// TIA Portal V15.1 export
// export: Created 2024-06-21T08:41:06.7682884Z, ExportSetting WithDefaults, DisplayName Totally Integrated Automation Portal, DisplayVersion V15.1 Update 5, DisplayName TIA Portal Openness, DisplayVersion V15.1 Update 5, DisplayName SINAMICS Startdrive Advanced, DisplayVersion V15.1, DisplayName G130, G150, S120, S150, SINAMICS MV, S210, DisplayVersion V15.1, DisplayName G110M, G120, G120C, G120D, G120P, DisplayVersion V15.1, DisplayName STEP 7 Professional, DisplayVersion V15.1 Update 5, DisplayName STEP 7 Safety, DisplayVersion V15.1, DisplayName WinCC Professional, DisplayVersion V15.1 Update 5, DisplayName SIMATIC Visualization Architect, DisplayVersion V15.1
FUNCTION_BLOCK "LGBBeltControl"   // FB6632, FBD
TITLE = LAcofDet / LGBBeltControl
{ S7_Optimized_Access := 'TRUE' }
AUTHOR : VCC
FAMILY : AlarmHandling
NAME : LGBBeltControl
VERSION : 1.0
// ===============================================================================
// This module handles a partdetection with all his functions and alarms
// Functions are DetCheckOn, DetCheckOff and EnableAlarm
// Outputs are DetAlarm and DetSim signal
// ===============================================================================
// ============================================================================
// This module handles Belt Slip Control
// ============================================================================
// stored: AutoNumber false, IsIECCheckEnabled false, IsRetainMemResEnabled false, MemoryReserve 100, SetENOAutomatically False, UDAEnableTagReadback false
   VAR_INPUT
      I_Det1SlipCtrl { ExternalAccessible := 'False'; ExternalVisible := 'False'; ExternalWritable := 'False'} : Bool;   // Actual input from sensor
      I_Det2SlipCtrl { ExternalAccessible := 'False'; ExternalVisible := 'False'; ExternalWritable := 'False'} : Bool;   // Actual input from sensor
      I_MotorRunning { ExternalAccessible := 'False'; ExternalVisible := 'False'; ExternalWritable := 'False'} : Bool;   // Previous detection
      I_EnableAlarm { ExternalAccessible := 'False'; ExternalVisible := 'False'; ExternalWritable := 'False'} : Bool;   // Enable Alarm
      I_AlarmClass { ExternalAccessible := 'False'; ExternalVisible := 'False'; ExternalWritable := 'False'} : Char;   // Alarm class -> A - B - C - D or E
      I_AlarmResetPB { ExternalAccessible := 'False'; ExternalVisible := 'False'; ExternalWritable := 'False'} : Bool;   // Alarm reset pushbutton is activated
   END_VAR
   VAR_OUTPUT
      O_Alarm { ExternalAccessible := 'False'; ExternalVisible := 'False'; ExternalWritable := 'False'} : Bool;   // Detection ON too long alarm / Detection alarm
      O_AlarmABCondition { ExternalAccessible := 'False'; ExternalVisible := 'False'; ExternalWritable := 'False'} : Bool;   // Alarm AB condition
   END_VAR
   VAR_IN_OUT
      H_HMI : "H_HMI";   // H_HMI
      H_BeltControl : "H_GBBeltControl";   // H_KTLBeltSlipControl
      IO_Modes : "Modes";
   END_VAR
   VAR
      CounterSlipCtrl { ExternalAccessible := 'False'; ExternalVisible := 'False'; ExternalWritable := 'False'} : DInt;   // Counter Slip Control
      CounterSlipCtrlL { ExternalAccessible := 'False'; ExternalVisible := 'False'; ExternalWritable := 'False'} : DInt;   // Counter Slip Control Left
      CounterSlipCtrlR { ExternalAccessible := 'False'; ExternalVisible := 'False'; ExternalWritable := 'False'} : DInt;   // Counter Slip Control Right
      AbsCounterSlipCtrl { ExternalAccessible := 'False'; ExternalVisible := 'False'; ExternalWritable := 'False'} : DInt;   // ABS Counter Slip Control
      ResetCount { ExternalAccessible := 'False'; ExternalVisible := 'False'; ExternalWritable := 'False'} : Bool;   // Reset Counters
      AlarmCond { ExternalAccessible := 'False'; ExternalVisible := 'False'; ExternalWritable := 'False'} : Bool;   // Alarm condition / Static variable of O_DetAlarm
      AlarmCondNOCountL { ExternalAccessible := 'False'; ExternalVisible := 'False'; ExternalWritable := 'False'} : Bool;   // Alarm condition / Static variable of O_DetAlarm
      AlarmCondNOCountR { ExternalAccessible := 'False'; ExternalVisible := 'False'; ExternalWritable := 'False'} : Bool;   // Alarm condition / Static variable of O_DetAlarm
      AlarmCondNCCountL { ExternalAccessible := 'False'; ExternalVisible := 'False'; ExternalWritable := 'False'} : Bool;   // Alarm condition / Static variable of O_DetAlarm
      AlarmCondNCCountR { ExternalAccessible := 'False'; ExternalVisible := 'False'; ExternalWritable := 'False'} : Bool;   // Alarm condition / Static variable of O_DetAlarm
      Alarm { ExternalAccessible := 'False'; ExternalVisible := 'False'; ExternalWritable := 'False'} : Bool;   // Alarm / Alarm condition
      AlarmClass_A { ExternalAccessible := 'False'; ExternalVisible := 'False'; ExternalWritable := 'False'} : Bool;   // The alarm is from alarm class A
      AlarmClass_B { ExternalAccessible := 'False'; ExternalVisible := 'False'; ExternalWritable := 'False'} : Bool;   // The alarm is from alarm class B
      AlarmClass_C { ExternalAccessible := 'False'; ExternalVisible := 'False'; ExternalWritable := 'False'} : Bool;   // The alarm is from alarm class C
      AlarmClass_D { ExternalAccessible := 'False'; ExternalVisible := 'False'; ExternalWritable := 'False'} : Bool;   // The alarm is from alarm class D
      AlarmClass_E { ExternalAccessible := 'False'; ExternalVisible := 'False'; ExternalWritable := 'False'} : Bool := false;   // The alarm is from alarm class E
      AlarmFiltered { ExternalAccessible := 'False'; ExternalVisible := 'False'; ExternalWritable := 'False'} : Bool;
      _TimerNoCountL { ExternalAccessible := 'False'; ExternalVisible := 'False'; ExternalWritable := 'False'} : "LTimer";
      _TimerNoCountR { ExternalAccessible := 'False'; ExternalVisible := 'False'; ExternalWritable := 'False'} : "LTimer";
      _TimerNcCountL { ExternalAccessible := 'False'; ExternalVisible := 'False'; ExternalWritable := 'False'} : "LTimer";
      _TimerNcCountR { ExternalAccessible := 'False'; ExternalVisible := 'False'; ExternalWritable := 'False'} : "LTimer";
      _TimerResetCount { ExternalAccessible := 'False'; ExternalVisible := 'False'; ExternalWritable := 'False'} : "LTimer";
      _TimerAlarmFilter { ExternalAccessible := 'False'; ExternalVisible := 'False'; ExternalWritable := 'False'} : "LTimer";
      edge { ExternalAccessible := 'False'; ExternalVisible := 'False'; ExternalWritable := 'False'} : Array[0..1] of Bool;
   END_VAR
   VAR_TEMP   // added for the SCL form of the ladder/FBD networks
      _w1 : Bool;
      _w2 : Bool;
   END_VAR
BEGIN

REGION Network 1: **** 1 - Inputs **** HMI Commands
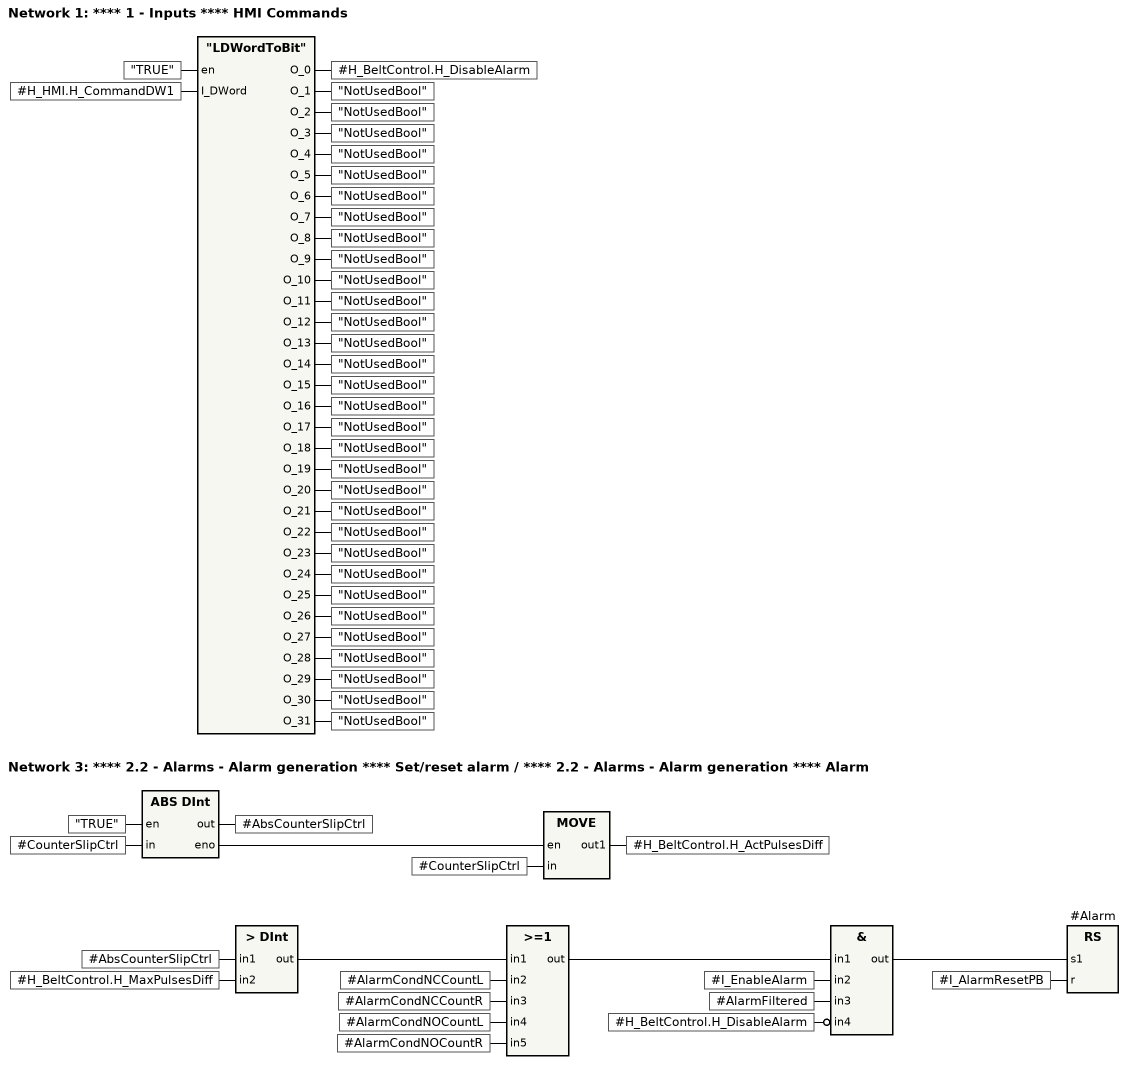
   IF "TRUE" THEN
       "LDWordToBit"(I_DWord := #H_HMI.H_CommandDW1,
                     O_0 => #H_BeltControl.H_DisableAlarm,
                     O_1 => "NotUsedBool",
                     O_2 => "NotUsedBool",
                     O_3 => "NotUsedBool",
                     O_4 => "NotUsedBool",
                     O_5 => "NotUsedBool",
                     O_6 => "NotUsedBool",
                     O_7 => "NotUsedBool",
                     O_8 => "NotUsedBool",
                     O_9 => "NotUsedBool",
                     O_10 => "NotUsedBool",
                     O_11 => "NotUsedBool",
                     O_12 => "NotUsedBool",
                     O_13 => "NotUsedBool",
                     O_14 => "NotUsedBool",
                     O_15 => "NotUsedBool",
                     O_16 => "NotUsedBool",
                     O_17 => "NotUsedBool",
                     O_18 => "NotUsedBool",
                     O_19 => "NotUsedBool",
                     O_20 => "NotUsedBool",
                     O_21 => "NotUsedBool",
                     O_22 => "NotUsedBool",
                     O_23 => "NotUsedBool",
                     O_24 => "NotUsedBool",
                     O_25 => "NotUsedBool",
                     O_26 => "NotUsedBool",
                     O_27 => "NotUsedBool",
                     O_28 => "NotUsedBool",
                     O_29 => "NotUsedBool",
                     O_30 => "NotUsedBool",
                     O_31 => "NotUsedBool");
   END_IF;
END_REGION

NETWORK
TITLE = **** 1 - Inputs **** Alarm class
// Alarm class
// Alarm class = E
      L     #I_AlarmClass;
      L     'E';
      ==I;
      =     #AlarmClass_E;

// Alarm class = D
      L     #I_AlarmClass;
      L     'D';
      ==I;
      =     #AlarmClass_D;

// Alarm class = C
      L     #I_AlarmClass;
      L     'C';
      ==I;
      =     #AlarmClass_C;

// Alarm class = B
      L     #I_AlarmClass;
      L     'B';
      ==I;
      =     #AlarmClass_B;

// Alarm class = A
      AN    #AlarmClass_B;
      AN    #AlarmClass_C;
      AN    #AlarmClass_D;
      AN    #AlarmClass_E;
      =     #AlarmClass_A;


REGION Network 3: **** 2.2 - Alarms - Alarm generation **** Set/reset alarm / **** 2.2 - Alarms - Alarm generation **** Alarm
   // Set/reset alarm
   IF "TRUE" THEN
       #AbsCounterSlipCtrl := ABS(#CounterSlipCtrl);
       #H_BeltControl.H_ActPulsesDiff := #CounterSlipCtrl;
   END_IF;
   IF #I_AlarmResetPB THEN
       #Alarm := FALSE;   // RS flip-flop
   END_IF;
   IF ((#AbsCounterSlipCtrl > #H_BeltControl.H_MaxPulsesDiff) OR #AlarmCondNCCountL OR #AlarmCondNCCountR OR #AlarmCondNOCountL OR #AlarmCondNOCountR) AND #I_EnableAlarm AND #AlarmFiltered AND NOT #H_BeltControl.H_DisableAlarm THEN
       #Alarm := TRUE;
   END_IF;
END_REGION

REGION Network 4: **** 2.2 - Alarms - Alarm generation **** Creating alarm overtime / **** 2.2 - Alarms - Alarm generation **** Pulses counters
   // Creating alarm overtime / Pulses counters
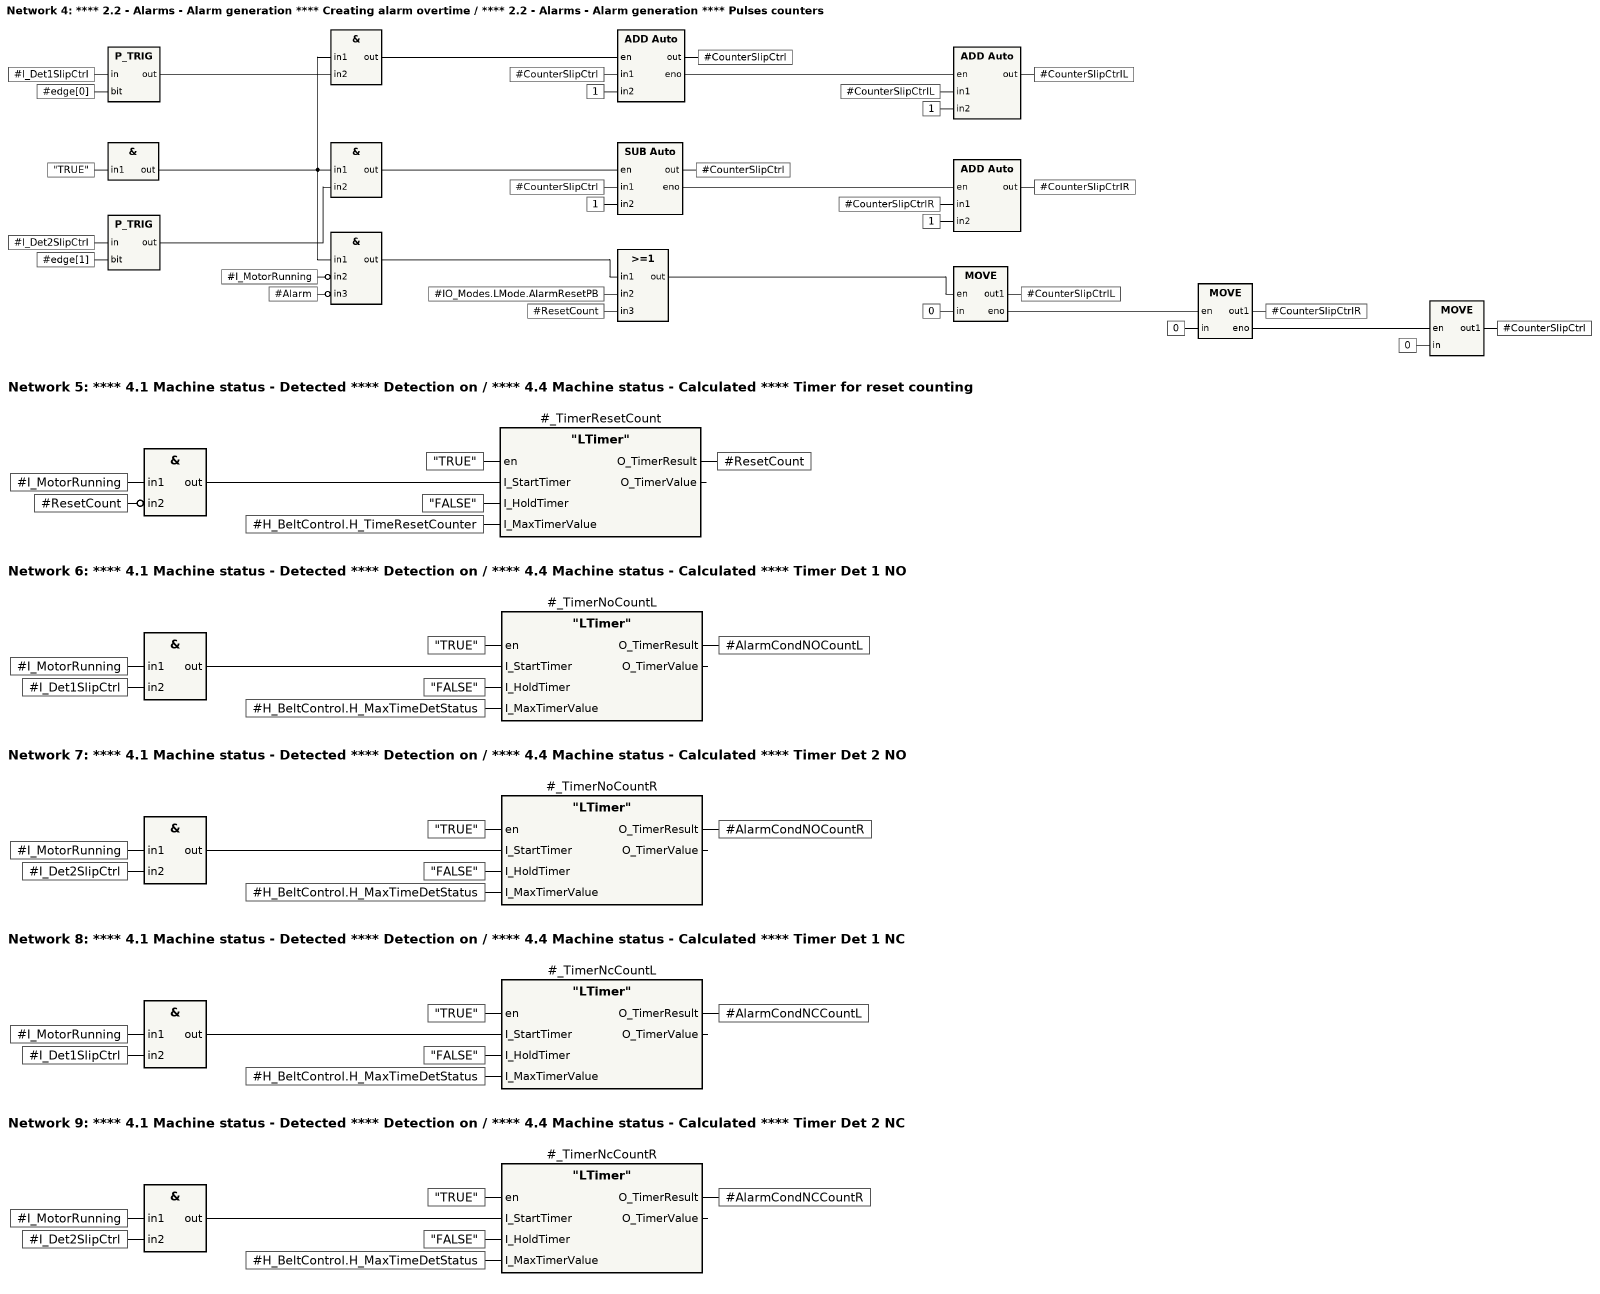
   #_w1 := #I_Det1SlipCtrl AND NOT #edge[0];   // rising edge
   #edge[0] := #I_Det1SlipCtrl;
   IF "TRUE" AND #_w1 THEN
       #CounterSlipCtrl := #CounterSlipCtrl + 1;
       #CounterSlipCtrlL := #CounterSlipCtrlL + 1;
   END_IF;
   #_w2 := #I_Det2SlipCtrl AND NOT #edge[1];   // rising edge
   #edge[1] := #I_Det2SlipCtrl;
   IF "TRUE" AND #_w2 THEN
       #CounterSlipCtrl := #CounterSlipCtrl - 1;
       #CounterSlipCtrlR := #CounterSlipCtrlR + 1;
   END_IF;
   IF ("TRUE" AND NOT #I_MotorRunning AND NOT #Alarm) OR #IO_Modes.LMode.AlarmResetPB OR #ResetCount THEN
       #CounterSlipCtrlL := 0;
       #CounterSlipCtrlR := 0;
       #CounterSlipCtrl := 0;
   END_IF;
END_REGION

REGION Network 5: **** 4.1 Machine status - Detected **** Detection on / **** 4.4 Machine status - Calculated **** Timer for reset counting
   // Detection on / Timer for reset counting
   IF "TRUE" THEN
       #_TimerResetCount(I_StartTimer := #I_MotorRunning AND NOT #ResetCount,   // "LTimer"
                         I_HoldTimer := "FALSE",
                         I_MaxTimerValue := #H_BeltControl.H_TimeResetCounter,
                         O_TimerResult => #ResetCount);
   END_IF;
END_REGION

REGION Network 6: **** 4.1 Machine status - Detected **** Detection on / **** 4.4 Machine status - Calculated **** Timer Det 1 NO
   // Detection on / Timer Det 1 NO
   IF "TRUE" THEN
       #_TimerNoCountL(I_StartTimer := #I_MotorRunning AND #I_Det1SlipCtrl,   // "LTimer"
                       I_HoldTimer := "FALSE",
                       I_MaxTimerValue := #H_BeltControl.H_MaxTimeDetStatus,
                       O_TimerResult => #AlarmCondNOCountL);
   END_IF;
END_REGION

REGION Network 7: **** 4.1 Machine status - Detected **** Detection on / **** 4.4 Machine status - Calculated **** Timer Det 2 NO
   // Detection on / Timer Det 2 NO
   IF "TRUE" THEN
       #_TimerNoCountR(I_StartTimer := #I_MotorRunning AND #I_Det2SlipCtrl,   // "LTimer"
                       I_HoldTimer := "FALSE",
                       I_MaxTimerValue := #H_BeltControl.H_MaxTimeDetStatus,
                       O_TimerResult => #AlarmCondNOCountR);
   END_IF;
END_REGION

REGION Network 8: **** 4.1 Machine status - Detected **** Detection on / **** 4.4 Machine status - Calculated **** Timer Det 1 NC
   // Detection on / Timer Det 1 NC
   IF "TRUE" THEN
       #_TimerNcCountL(I_StartTimer := #I_MotorRunning AND #I_Det1SlipCtrl,   // "LTimer"
                       I_HoldTimer := "FALSE",
                       I_MaxTimerValue := #H_BeltControl.H_MaxTimeDetStatus,
                       O_TimerResult => #AlarmCondNCCountL);
   END_IF;
END_REGION

REGION Network 9: **** 4.1 Machine status - Detected **** Detection on / **** 4.4 Machine status - Calculated **** Timer Det 2 NC
   // Detection on / Timer Det 2 NC
   IF "TRUE" THEN
       #_TimerNcCountR(I_StartTimer := #I_MotorRunning AND #I_Det2SlipCtrl,   // "LTimer"
                       I_HoldTimer := "FALSE",
                       I_MaxTimerValue := #H_BeltControl.H_MaxTimeDetStatus,
                       O_TimerResult => #AlarmCondNCCountR);
   END_IF;
END_REGION

REGION Network 10: **** 4.1 Machine status - Detected **** Detection on / **** 4.4 Machine status - Calculated **** Timer Alarm Filter
   // Detection on / Timer Det 2 NC
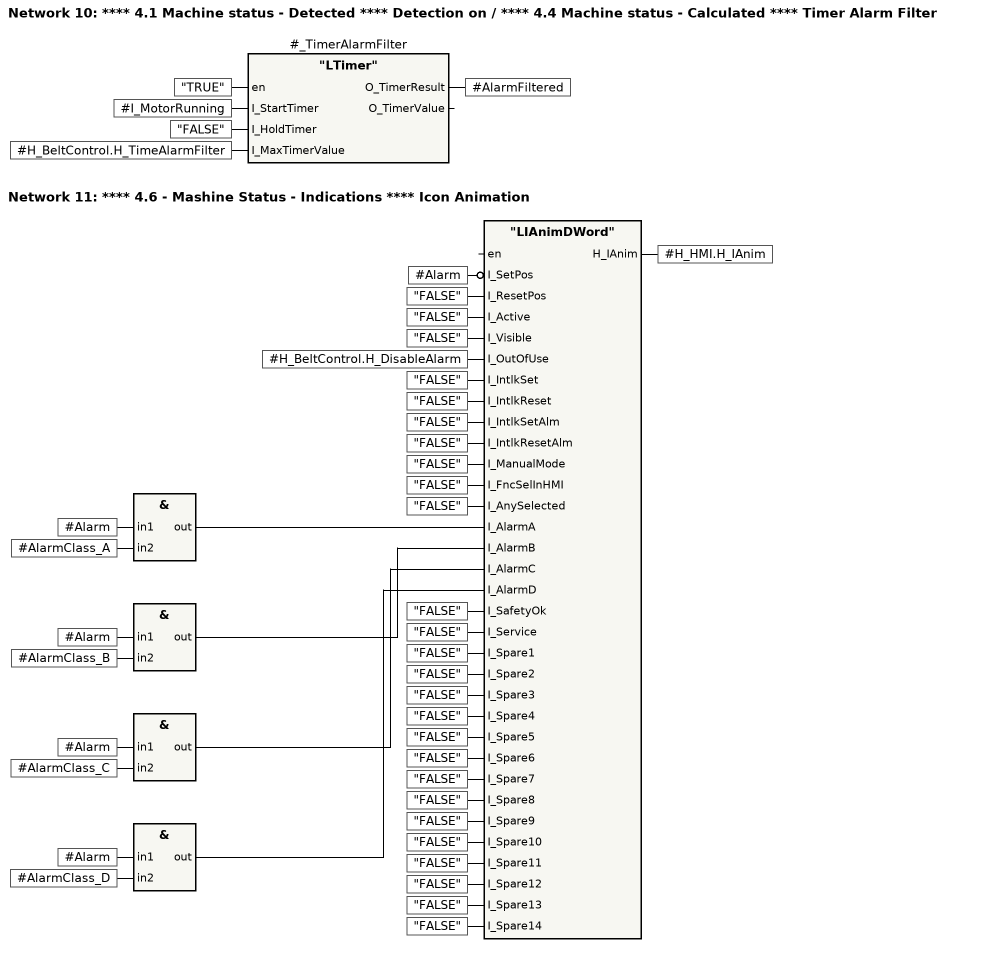
   IF "TRUE" THEN
       #_TimerAlarmFilter(I_StartTimer := #I_MotorRunning,   // "LTimer"
                          I_HoldTimer := "FALSE",
                          I_MaxTimerValue := #H_BeltControl.H_TimeAlarmFilter,
                          O_TimerResult => #AlarmFiltered);
   END_IF;
END_REGION

REGION Network 11: **** 4.6 - Mashine Status - Indications **** Icon Animation
   // Icon Animation
   "LIAnimDWord"(I_SetPos := NOT #Alarm,
                 I_ResetPos := "FALSE",
                 I_Active := "FALSE",
                 I_Visible := "FALSE",
                 I_OutOfUse := #H_BeltControl.H_DisableAlarm,
                 I_IntlkSet := "FALSE",
                 I_IntlkReset := "FALSE",
                 I_IntlkSetAlm := "FALSE",
                 I_IntlkResetAlm := "FALSE",
                 I_ManualMode := "FALSE",
                 I_FncSelInHMI := "FALSE",
                 I_AnySelected := "FALSE",
                 I_AlarmA := #Alarm AND #AlarmClass_A,
                 I_AlarmB := #Alarm AND #AlarmClass_B,
                 I_AlarmC := #Alarm AND #AlarmClass_C,
                 I_AlarmD := #Alarm AND #AlarmClass_D,
                 I_SafetyOk := "FALSE",
                 I_Service := "FALSE",
                 I_Spare1 := "FALSE",
                 I_Spare2 := "FALSE",
                 I_Spare3 := "FALSE",
                 I_Spare4 := "FALSE",
                 I_Spare5 := "FALSE",
                 I_Spare6 := "FALSE",
                 I_Spare7 := "FALSE",
                 I_Spare8 := "FALSE",
                 I_Spare9 := "FALSE",
                 I_Spare10 := "FALSE",
                 I_Spare11 := "FALSE",
                 I_Spare12 := "FALSE",
                 I_Spare13 := "FALSE",
                 I_Spare14 := "FALSE",
                 H_IAnim => #H_HMI.H_IAnim);
END_REGION

REGION Network 12: **** 4.6 - Machine Status - Indications **** Animation
   // Animation
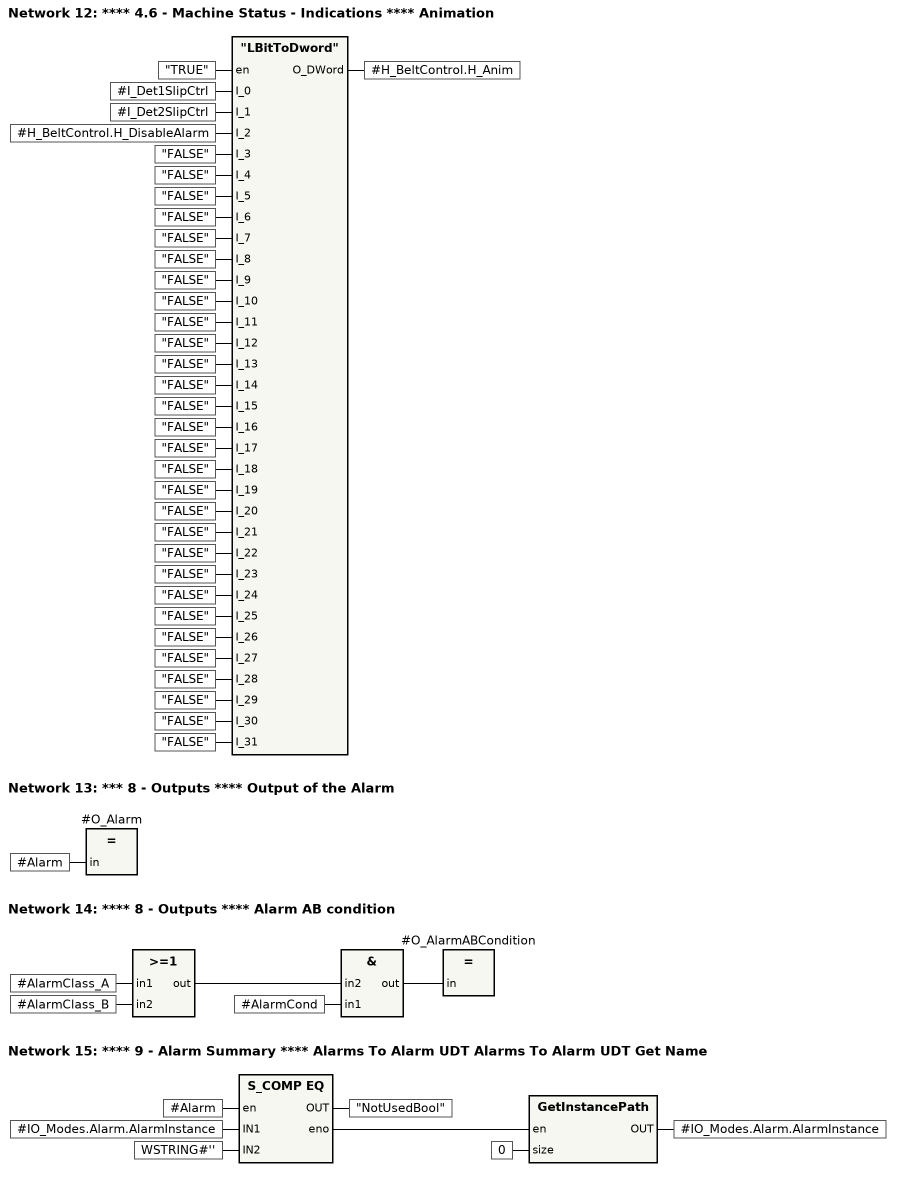
   IF "TRUE" THEN
       "LBitToDword"(I_0 := #I_Det1SlipCtrl,
                     I_1 := #I_Det2SlipCtrl,
                     I_2 := #H_BeltControl.H_DisableAlarm,
                     I_3 := "FALSE",
                     I_4 := "FALSE",
                     I_5 := "FALSE",
                     I_6 := "FALSE",
                     I_7 := "FALSE",
                     I_8 := "FALSE",
                     I_9 := "FALSE",
                     I_10 := "FALSE",
                     I_11 := "FALSE",
                     I_12 := "FALSE",
                     I_13 := "FALSE",
                     I_14 := "FALSE",
                     I_15 := "FALSE",
                     I_16 := "FALSE",
                     I_17 := "FALSE",
                     I_18 := "FALSE",
                     I_19 := "FALSE",
                     I_20 := "FALSE",
                     I_21 := "FALSE",
                     I_22 := "FALSE",
                     I_23 := "FALSE",
                     I_24 := "FALSE",
                     I_25 := "FALSE",
                     I_26 := "FALSE",
                     I_27 := "FALSE",
                     I_28 := "FALSE",
                     I_29 := "FALSE",
                     I_30 := "FALSE",
                     I_31 := "FALSE",
                     O_DWord => #H_BeltControl.H_Anim);
   END_IF;
END_REGION

REGION Network 13: *** 8 - Outputs **** Output of the Alarm
   // Output of the Alarm
   #O_Alarm := #Alarm;
END_REGION

REGION Network 14: **** 8 - Outputs **** Alarm AB condition
   // Alarm AB condition
   #O_AlarmABCondition := (#AlarmClass_A OR #AlarmClass_B) AND #AlarmCond;
END_REGION

REGION Network 15: **** 9 - Alarm Summary **** Alarms To Alarm UDT Alarms To Alarm UDT Get Name
   // Alarm / Alarm D
   S_COMP(EN := #Alarm,
          IN1 := #IO_Modes.Alarm.AlarmInstance,
          IN2 := WSTRING#'',
          OUT => "NotUsedBool",
          ENO => #_w1);
   IF #_w1 THEN GetInstancePath(size := 0, OUT => #IO_Modes.Alarm.AlarmInstance); END_IF;
END_REGION

REGION Network 16: **** 9 - Alarm Summary **** Alarms To Alarm UDT
   // Alarm / Alarm D
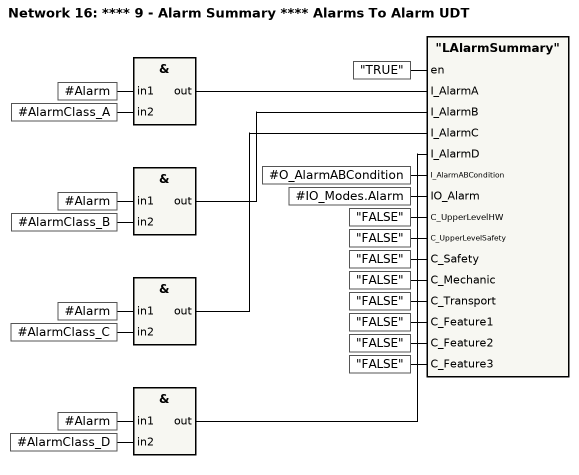
   IF "TRUE" THEN
       "LAlarmSummary"(I_AlarmA := #Alarm AND #AlarmClass_A,
                       I_AlarmB := #Alarm AND #AlarmClass_B,
                       I_AlarmC := #Alarm AND #AlarmClass_C,
                       I_AlarmD := #Alarm AND #AlarmClass_D,
                       I_AlarmABCondition := #O_AlarmABCondition,
                       IO_Alarm := #IO_Modes.Alarm,
                       C_UpperLevelHW := "FALSE",
                       C_UpperLevelSafety := "FALSE",
                       C_Safety := "FALSE",
                       C_Mechanic := "FALSE",
                       C_Transport := "FALSE",
                       C_Feature1 := "FALSE",
                       C_Feature2 := "FALSE",
                       C_Feature3 := "FALSE");
   END_IF;
END_REGION
END_FUNCTION_BLOCK
